(* Logix 5000 project; controller EuniceF_ICA12 vendor 1 type 14 code 150 rev 37.11; software revision 37.00 *)

TASK MainTask (continuous, watchdog 500 ms) : MainProgram

MODULES
   Local : vendor 1 type 14 code 150 (Compact 0, rev 37.11)
      Discrete_IO : Embedded (Compact 1, rev 3.1, Output RPI 20 ms)
      Analog_IO : Embedded (Compact 2, rev 1.1, Output RPI 80 ms)
      Counters : Embedded (Compact 3, rev 1.1, Output RPI 20 ms)
END_MODULES

VAR_GLOBAL   (* controller tags *)
   M1 : ALIAS FOR Local:1:O.Data.4;
   M2 : ALIAS FOR Local:1:O.Data.5;
   M3 : ALIAS FOR Local:1:O.Data.6;
   MOTOR : ALIAS FOR Local:1:O.Data.1;
   MOTOR1 : ALIAS FOR Local:1:O.Data.1;
   MOTOR2 : ALIAS FOR Local:1:O.Data.2;
   MOTOR3 : ALIAS FOR Local:1:O.Data.3;
   START : ALIAS FOR Local:1:I.Data.11;
   START1 : ALIAS FOR Local:1:I.Data.12;
   STOP : ALIAS FOR Local:1:I.Data.8;
   STOP1 : ALIAS FOR Local:1:I.Data.9;
   T1 : TIMER := (PRE := 2000);
   T2 : TIMER := (PRE := 4000);
   T_STOP : TIMER := (PRE := 3000);
   T_stop1 : TIMER := (PRE := 3000);
   Timer1 : TIMER := (PRE := 5000);
   TIMER2 : TIMER := (PRE := 3000);
   TSTOP : BOOL;
END_VAR

PROGRAM MainProgram   (* main routine MainRoutine *)

ROUTINE MainRoutine   (* ladder *)
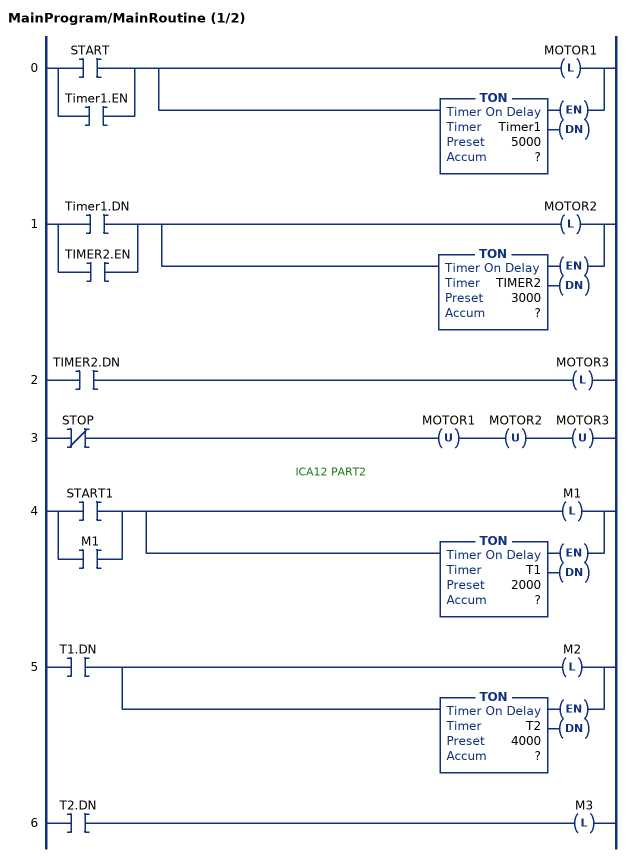
   0: [XIC(START) ,XIC(Timer1.EN) ][OTL(MOTOR1) ,TON(Timer1,?,?) ];
   1: [XIC(Timer1.DN) ,XIC(TIMER2.EN) ][OTL(MOTOR2) ,TON(TIMER2,?,?) ];
   2: XIC(TIMER2.DN)OTL(MOTOR3);
   3: XIO(STOP)OTU(MOTOR1)OTU(MOTOR2)OTU(MOTOR3);
   // ICA12 PART2
   4: [XIC(START1) ,XIC(M1) ][OTL(M1) ,TON(T1,?,?) ];
   5: XIC(T1.DN)[OTL(M2) ,TON(T2,?,?) ];
   6: XIC(T2.DN)OTL(M3);
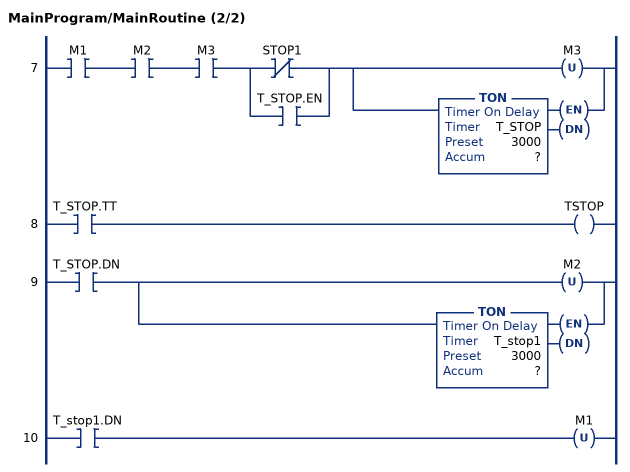
   7: XIC(M1)XIC(M2)XIC(M3)[XIO(STOP1) ,XIC(T_STOP.EN) ][OTU(M3) ,TON(T_STOP,?,?) ];
   8 (stored rung type 13): XIC(T_STOP.TT)OTE(TSTOP);
   9: XIC(T_STOP.DN)[OTU(M2) ,TON(T_stop1,?,?) ];
   10: XIC(T_stop1.DN)OTU(M1);
END_ROUTINE
END_PROGRAM
